Staubli VAL3: VelocityCmd.dtx

public num nSeq
public num nVelVec[6]
public num nCmdType
